TYPE U_TICKET_LIST_DATA_OUTPUT :
UNION
  stData              : ST_LIST_NODE_DATA;
  byData   AT %Q*     : ARRAY[1..SIZEOF(ST_LIST_NODE_DATA)] OF BYTE;
END_UNION
END_TYPE

(* stored: Version 1.1.0.1, ProductVersion 3.1.4026.13
   DUT U_TICKET_LIST_DATA_OUTPUT: Id {ef70b86d-d661-4b75-8662-be6e82158157} *)
